RoboDK station: tst_square.rdk

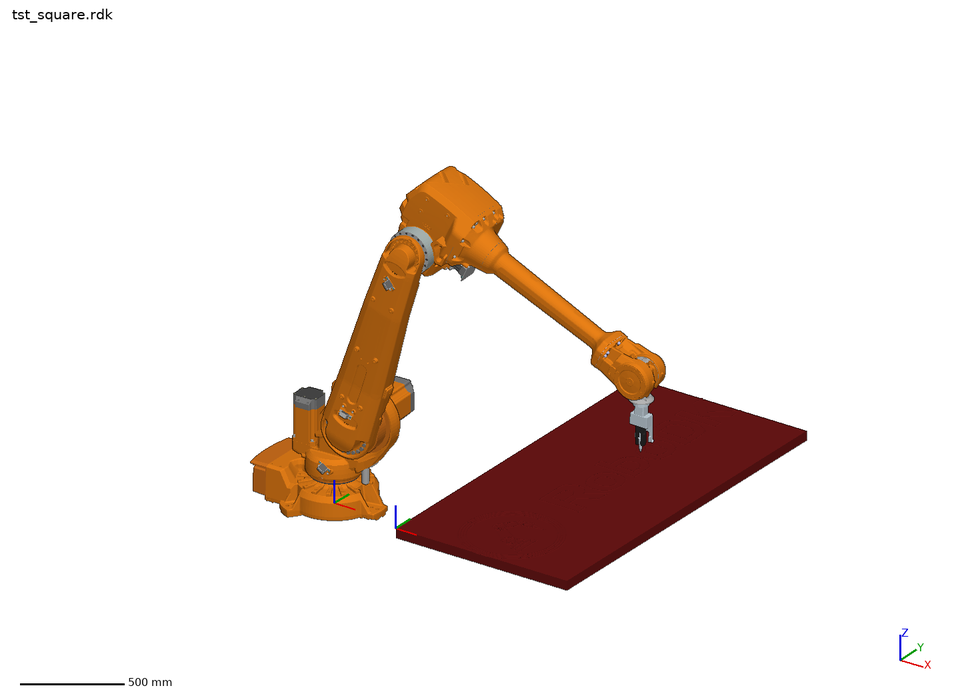
[picture v0: the station drawn from its stored meshes, robots at their saved joint values, targets as dots, program paths as lines]
Station tst_square (saved by RoboDK 5.6.3). Poses are relative to the parent item; angles as X-Y-Z fixed-axis rotations.
Station parameters (name, value as stored): TAGS, ['Drawing']
  - frame ABB IRB 4600-20/2.50 Base at (0, 0, 0) mm
    - robot ABB IRB 4600-20/2.50: 6 axes, payload 20 kg, reach 2500 mm, repeatability 0.05 mm, weight 412 kg
        modified DH rows (alpha deg, a mm, theta deg, d mm): 0, 0, 0, 495; -90, 175, -90, 0; 0, 1095, 0, 0; -90, 175, 0, 1270; 90, 0, 0, 0; -90, 0, 180, 135
        joint limits [-180, -90, -180, -400, -120, -400] to [180, 150, 75, 400, 120, 400]; home [0, 0, 0, 0, 90, 0]; saved at [2.34, 18.53, 6.85, 0.01, 65.54, 1.85]
      - tool Tool, TCP at (0, 0, 283) mm, size 100 x 89.2 x 281.5 mm
    - object pixel at (0, 0, 0) mm, size 10 x 10 x 1 mm
    - frame Draw Frame at (1016.5, -940.57, 525.71) mm
      - object Whiteboard 250mm at (0, 0, 0) mm, size 250 x 250 x 50 mm
      - object Drawing Board at (0, 0, 0) mm, size 1000 x 2011.6 x 51 mm
  - Python program square (listed below)

--- Python program square ---
from robodk.robolink import *
from robodk.robomath import *

# Any interaction with RoboDK must be done through RDK:
RDK = Robolink()

# Select a robot (popup is displayed if more than one robot is available)
robot = RDK.ItemUserPick('Select a robot', ITEM_TYPE_ROBOT)
if not robot.Valid():
    raise Exception('No robot selected or available')

# Get the current position of the TCP with respect to the reference frame:
# (4x4 matrix representing position and orientation)
target_ref = robot.Pose()
pos_ref = target_ref.Pos()
print("Drawing a square around the target: ")
print(Pose_2_TxyzRxyz(target_ref))

# Move the robot to the first point:
robot.MoveJ(target_ref)

# It is important to provide the reference frame and the tool frames when generating programs offline
robot.setPoseFrame(robot.PoseFrame())
robot.setPoseTool(robot.PoseTool())
robot.setRounding(10)  # Set the rounding parameter
robot.setSpeed(50)   # Set linear speed in mm/s

# Set the number of sides of the polygon (for a square, it's 4):
n_sides = 5
side_length = 500  # 3 cm in mm


def draw_box(edges):
    for edge in edges:
        target_i = Mat(target_ref)
        pos_i = target_i.Pos()
        print("target_i", target_i)
        print("pos_i before change :",pos_i)

        pos_i[0] = pos_i[0] + edge[0]
        pos_i[1] = pos_i[1] + edge[1]
        pos_i[2] = pos_i[2] - 200


        target_i.setPos(pos_i)
        # print("Moving to target %i: angle %.1f" % (i, ang * 180 / pi))
        print(str(Pose_2_TxyzRxyz(target_i)))
        robot.MoveL(target_i)

    target_i = Mat(target_ref)
    pos_i = target_i.Pos()
    pos_i[0] = pos_i[0] + edges[0][0]
    pos_i[1] = pos_i[1] + edges[0][1]
    pos_i[2] = pos_i[2] -200
    target_i.setPos(pos_i)
    robot.MoveL(target_i)

    robot.MoveL(target_ref)



if __name__ == "__main__":
    edges = [
        [0,0],
        [250,0],
        [250,550],
        [0,550]
    ]
    draw_box(edges)
print('Done')
